// TIA Portal V16 export
// export: Created 2021-05-25T16:14:34.663981Z, ExportSetting WithDefaults, DisplayName Totally Integrated Automation Portal, DisplayVersion V16, DisplayName TIA Portal Version Control Interface, DisplayVersion V16, DisplayName TIA Portal Openness, DisplayVersion V16, DisplayName STEP 7 Professional, DisplayVersion V16, DisplayName STEP 7 Safety, DisplayVersion V16, DisplayName WinCC Unified SCADA Engineering System, DisplayVersion V16
DATA_BLOCK "ph_Helix_1_DB"   // DB310
VERSION : 0.1
// stored: AutoNumber false, DBAccessibleFromOPCUA true, InstanceOfName ph_Helix_1, InstanceOfType FB
"ph_Helix_1"
   // VAR_IN_OUT
   //    Y8_VijaLocev_Des : "udtDigitalValve";
   //    Y9_VijaStop_DesZad : "udtDigitalValve";
   //    Y2_VijaDesZad_Dvig : "udtDigitalValve";
   //    Y10_Centri_DesZad : "udtDigitalValve";
   //    Y3_VijaDesSpr_Dvig : "udtDigitalValve";
   //    Y11_Centri_DesSpr : "udtDigitalValve";
   //    Y12_VijaLocev_Lev : "udtDigitalValve";
   //    Y13_VijaStop_LevZad : "udtDigitalValve";
   //    Y4_VijaLevZad_Dvig : "udtDigitalValve";
   //    Y14_Centri_LevZad : "udtDigitalValve";
   //    Y5_VijaLevSpr_Dvig : "udtDigitalValve";
   //    Y15_Centri_LevSpr : "udtDigitalValve";
   //    Y16_VpenjanjeDna : "udtDigitalValve";
   //    M1_ZADAJ_LEVO : "udtMotor";
   //    M2_SPREDAJ_LEVO : "udtMotor";
   //    M1_ZADAJ_DESNO : "udtMotor";
   //    M2_SPREDAJ_DESNO : "udtMotor";
   //    VKLOP_M_TRAKA_VIJACNIKA : "udtMotor";
   // END_VAR
   // VAR RETAIN
   //    CurrentStep { ExternalAccessible := 'False'; ExternalVisible := 'False'; ExternalWritable := 'False'} : Int := 10;
   //    PhaseStatus { ExternalAccessible := 'False'; ExternalVisible := 'False'; ExternalWritable := 'False'} : Int := 5;
   // END_VAR
   // VAR
   //    AlarmPresent { ExternalAccessible := 'False'; ExternalVisible := 'False'; ExternalWritable := 'False'} : Bool := FALSE;
   //    InitPosition { ExternalAccessible := 'False'; ExternalVisible := 'False'; ExternalWritable := 'False'} : Bool := TRUE;
   //    StartCmd { ExternalAccessible := 'False'; ExternalVisible := 'False'; ExternalWritable := 'False'} : Bool := TRUE;
   //    AlarmPresentOLD { ExternalAccessible := 'False'; ExternalVisible := 'False'; ExternalWritable := 'False'} : Bool := FALSE;
   //    InitPositionOLD { ExternalAccessible := 'False'; ExternalVisible := 'False'; ExternalWritable := 'False'} : Bool := TRUE;
   //    IEC_TimerOnDly_1 { ExternalAccessible := 'False'; ExternalVisible := 'False'; ExternalWritable := 'False'} : TONR_TIME;
   //    IEC_TimerOnDly_2 { ExternalAccessible := 'False'; ExternalVisible := 'False'; ExternalWritable := 'False'} : TONR_TIME;
   //    IEC_TimerOnDly_3 { ExternalAccessible := 'False'; ExternalVisible := 'False'; ExternalWritable := 'False'} : TONR_TIME;
   //    IEC_TimerOnDly_4 { ExternalAccessible := 'False'; ExternalVisible := 'False'; ExternalWritable := 'False'} : TONR_TIME;
   //    IEC_TimerOnDly_5 { ExternalAccessible := 'False'; ExternalVisible := 'False'; ExternalWritable := 'False'} : TONR_TIME;
   //    IEC_TimerOnDly_6 { ExternalAccessible := 'False'; ExternalVisible := 'False'; ExternalWritable := 'False'} : TONR_TIME;
   //    IEC_TimerOnDly_7 { ExternalAccessible := 'False'; ExternalVisible := 'False'; ExternalWritable := 'False'} : TONR_TIME;
   //    IEC_TimerOnDly_8 { ExternalAccessible := 'False'; ExternalVisible := 'False'; ExternalWritable := 'False'} : TONR_TIME;
   //    IEC_TimerOnDly_9 { ExternalAccessible := 'False'; ExternalVisible := 'False'; ExternalWritable := 'False'} : TONR_TIME;
   //    IEC_TimerOnDly_10 { ExternalAccessible := 'False'; ExternalVisible := 'False'; ExternalWritable := 'False'} : TONR_TIME;
   //    IEC_TimerOnDly_ET_1 { ExternalAccessible := 'False'; ExternalVisible := 'False'; ExternalWritable := 'False'} : Time := T#0MS;
   //    IEC_TimerOnDly_ET_2 { ExternalAccessible := 'False'; ExternalVisible := 'False'; ExternalWritable := 'False'} : Time := T#0MS;
   //    IEC_TimerOnDly_ET_3 { ExternalAccessible := 'False'; ExternalVisible := 'False'; ExternalWritable := 'False'} : Time := T#0MS;
   //    IEC_TimerOnDly_ET_4 { ExternalAccessible := 'False'; ExternalVisible := 'False'; ExternalWritable := 'False'} : Time := T#0MS;
   //    IEC_TimerOnDly_ET_5 { ExternalAccessible := 'False'; ExternalVisible := 'False'; ExternalWritable := 'False'} : Time := T#0MS;
   //    IEC_TimerOnDly_ET_6 { ExternalAccessible := 'False'; ExternalVisible := 'False'; ExternalWritable := 'False'} : Time := T#0MS;
   //    IEC_TimerOnDly_ET_7 { ExternalAccessible := 'False'; ExternalVisible := 'False'; ExternalWritable := 'False'} : Time := T#0MS;
   //    IEC_TimerOnDly_ET_8 { ExternalAccessible := 'False'; ExternalVisible := 'False'; ExternalWritable := 'False'} : Time := T#0MS;
   //    IEC_TimerOnDly_ET_9 { ExternalAccessible := 'False'; ExternalVisible := 'False'; ExternalWritable := 'False'} : Time := T#0MS;
   //    IEC_TimerOnDly_ET_10 { ExternalAccessible := 'False'; ExternalVisible := 'False'; ExternalWritable := 'False'} : Time := T#0MS;
   //    IEC_TimerOnDly_DN_1 { ExternalAccessible := 'False'; ExternalVisible := 'False'; ExternalWritable := 'False'} : Bool := FALSE;
   //    IEC_TimerOnDly_DN_2 { ExternalAccessible := 'False'; ExternalVisible := 'False'; ExternalWritable := 'False'} : Bool := FALSE;
   //    IEC_TimerOnDly_DN_3 { ExternalAccessible := 'False'; ExternalVisible := 'False'; ExternalWritable := 'False'} : Bool := FALSE;
   //    IEC_TimerOnDly_DN_4 { ExternalAccessible := 'False'; ExternalVisible := 'False'; ExternalWritable := 'False'} : Bool := FALSE;
   //    IEC_TimerOnDly_DN_5 { ExternalAccessible := 'False'; ExternalVisible := 'False'; ExternalWritable := 'False'} : Bool := FALSE;
   //    IEC_TimerOnDly_DN_6 { ExternalAccessible := 'False'; ExternalVisible := 'False'; ExternalWritable := 'False'} : Bool := FALSE;
   //    IEC_TimerOnDly_DN_7 { ExternalAccessible := 'False'; ExternalVisible := 'False'; ExternalWritable := 'False'} : Bool := FALSE;
   //    IEC_TimerOnDly_DN_8 { ExternalAccessible := 'False'; ExternalVisible := 'False'; ExternalWritable := 'False'} : Bool := FALSE;
   //    IEC_TimerOnDly_DN_9 { ExternalAccessible := 'False'; ExternalVisible := 'False'; ExternalWritable := 'False'} : Bool := FALSE;
   //    IEC_TimerOnDly_DN_10 { ExternalAccessible := 'False'; ExternalVisible := 'False'; ExternalWritable := 'False'} : Bool := FALSE;
   //    LeftLegIndex { ExternalAccessible := 'False'; ExternalVisible := 'False'; ExternalWritable := 'False'} : Int := 2;
   //    RightLegIndex { ExternalAccessible := 'False'; ExternalVisible := 'False'; ExternalWritable := 'False'} : Int := 2;
   //    LeftLegsArrayIndex { ExternalAccessible := 'False'; ExternalVisible := 'False'; ExternalWritable := 'False'} : Array[1..6] of Bool;
   //    RightLegsArrayIndex { ExternalAccessible := 'False'; ExternalVisible := 'False'; ExternalWritable := 'False'} : Array[1..6] of Bool;
   //    ButtomFasting_Activated { ExternalAccessible := 'False'; ExternalVisible := 'False'; ExternalWritable := 'False'} : Bool := TRUE;
   //    Helix_Activated { ExternalAccessible := 'False'; ExternalVisible := 'False'; ExternalWritable := 'False'} : Bool := FALSE;
   // END_VAR
   // VAR RETAIN
   //    DlyToFinishButtonFasten { S7_SetPoint := 'True'} : Int := 2;
   // END_VAR
   // VAR
   //    MovingUPDOWN_Activated { ExternalAccessible := 'False'; ExternalVisible := 'False'; ExternalWritable := 'False'} : Bool := FALSE;
   //    MoveUPDOWN_LevoSpredaj { ExternalAccessible := 'False'; ExternalVisible := 'False'; ExternalWritable := 'False'} : Bool := FALSE;
   //    MoveUPDOWN_LevoZadaj { ExternalAccessible := 'False'; ExternalVisible := 'False'; ExternalWritable := 'False'} : Bool := FALSE;
   //    MoveUPDOWN_DESNOSpredaj { ExternalAccessible := 'False'; ExternalVisible := 'False'; ExternalWritable := 'False'} : Bool := FALSE;
   //    MoveUPDOWN_DESNOZadaj { ExternalAccessible := 'False'; ExternalVisible := 'False'; ExternalWritable := 'False'} : Bool := FALSE;
   // END_VAR
   // VAR RETAIN
   //    DlyToRotateOpposite { S7_SetPoint := 'True'} : Int := 10;
   //    WaitTimeBeforeMoveDown { S7_SetPoint := 'True'} : Int := 2;
   // END_VAR
   // VAR
   //    WaitLevoSpredaj { ExternalAccessible := 'False'; ExternalVisible := 'False'; ExternalWritable := 'False'} : Bool := FALSE;
   //    WaitLevoZadaj { ExternalAccessible := 'False'; ExternalVisible := 'False'; ExternalWritable := 'False'} : Bool := FALSE;
   //    WaitDesnoSpredaj { ExternalAccessible := 'False'; ExternalVisible := 'False'; ExternalWritable := 'False'} : Bool := FALSE;
   //    WaitDesnoZadaj { ExternalAccessible := 'False'; ExternalVisible := 'False'; ExternalWritable := 'False'} : Bool := FALSE;
   //    FOTOCELICA_LOC_TRAK_LEVO1_Latch { ExternalAccessible := 'False'; ExternalVisible := 'False'; ExternalWritable := 'False'} : Bool := FALSE;
   //    FOTOCELICA_LOC_TRAK_LEVO2_Latch { ExternalAccessible := 'False'; ExternalVisible := 'False'; ExternalWritable := 'False'} : Bool := FALSE;
   //    FOTOCELICA_LOC_TRAK_DESNO1_Latch { ExternalAccessible := 'False'; ExternalVisible := 'False'; ExternalWritable := 'False'} : Bool := FALSE;
   //    FOTOCELICA_LOC_TRAK_DESNO2_Latch { ExternalAccessible := 'False'; ExternalVisible := 'False'; ExternalWritable := 'False'} : Bool := FALSE;
   // END_VAR
   // VAR RETAIN
   //    WEndTimeToRemovePlate { S7_SetPoint := 'True'} : Int := 2;
   // END_VAR
   // VAR
   //    LeftLegIndexOLD { ExternalAccessible := 'False'; ExternalVisible := 'False'; ExternalWritable := 'False'} : Int := 2;
   //    RightLegIndexOLD { ExternalAccessible := 'False'; ExternalVisible := 'False'; ExternalWritable := 'False'} : Int := 2;
   //    StartReleaseTimer1 { ExternalAccessible := 'False'; ExternalVisible := 'False'; ExternalWritable := 'False'} : Bool := FALSE;
   //    StartReleaseTimer2 { ExternalAccessible := 'False'; ExternalVisible := 'False'; ExternalWritable := 'False'} : Bool := FALSE;
   //    FOTOCELICA_LEVO_SPREDAJ_LATCH { ExternalAccessible := 'False'; ExternalVisible := 'False'; ExternalWritable := 'False'} : Bool := TRUE;
   //    FOTOCELICA_LEVO_ZADAJ_LATCH { ExternalAccessible := 'False'; ExternalVisible := 'False'; ExternalWritable := 'False'} : Bool := TRUE;
   //    FOTOCELICA_DESNO_SPREDAJ_LATCH { ExternalAccessible := 'False'; ExternalVisible := 'False'; ExternalWritable := 'False'} : Bool := TRUE;
   //    FOTOCELICA_DESNO_ZADAJ_LATCH { ExternalAccessible := 'False'; ExternalVisible := 'False'; ExternalWritable := 'False'} : Bool := TRUE;
   // END_VAR
   // VAR RETAIN
   //    DlyToStartButtomFasten { S7_SetPoint := 'True'} : Int := 10;
   // END_VAR
   // VAR
   //    EndLevoSpredaj { ExternalAccessible := 'False'; ExternalVisible := 'False'; ExternalWritable := 'False'} : Bool := FALSE;
   //    EndLevoZadaj { ExternalAccessible := 'False'; ExternalVisible := 'False'; ExternalWritable := 'False'} : Bool := FALSE;
   //    EndDesnoSpredaj { ExternalAccessible := 'False'; ExternalVisible := 'False'; ExternalWritable := 'False'} : Bool := FALSE;
   //    EndDesnoZadaj { ExternalAccessible := 'False'; ExternalVisible := 'False'; ExternalWritable := 'False'} : Bool := FALSE;
   // END_VAR
   // VAR RETAIN
   //    DlyToInitRunTrakVijac { ExternalAccessible := 'False'; ExternalVisible := 'False'; ExternalWritable := 'False'; S7_SetPoint := 'True'} : Int := 20;
   // END_VAR
   // VAR
   //    LegsReadyOnPosToHelix { ExternalAccessible := 'False'; ExternalVisible := 'False'; ExternalWritable := 'False'} : Bool := FALSE;
   //    VpenjanjeDnaActived { ExternalAccessible := 'False'; ExternalVisible := 'False'; ExternalWritable := 'False'} : Bool := FALSE;
   // END_VAR
   // VAR RETAIN
   //    RegimeHelix { S7_SetPoint := 'True'} : Bool := TRUE;
   //    TotalButtomPlateCounter : UDInt := 4;
   // END_VAR
   // VAR
   //    DetectStartButtom { ExternalAccessible := 'False'; ExternalVisible := 'False'; ExternalWritable := 'False'} : Bool := FALSE;
   //    InsertNewButtom { ExternalAccessible := 'False'; ExternalVisible := 'False'; ExternalWritable := 'False'} : USInt := 1;
   // END_VAR
   // VAR RETAIN
   //    TimeoutToEndHelix { ExternalAccessible := 'False'; ExternalVisible := 'False'; ExternalWritable := 'False'; S7_SetPoint := 'True'} : UInt := 80;
   // END_VAR
   // VAR
   //    FirstButtom { ExternalAccessible := 'False'; ExternalVisible := 'False'; ExternalWritable := 'False'} : Bool := FALSE;
   // END_VAR
BEGIN
   IEC_TimerOnDly_1.PT := T#0MS;
   IEC_TimerOnDly_1.IN := FALSE;
   IEC_TimerOnDly_2.PT := T#0MS;
   IEC_TimerOnDly_2.IN := FALSE;
   IEC_TimerOnDly_3.PT := T#0MS;
   IEC_TimerOnDly_3.IN := FALSE;
   IEC_TimerOnDly_4.PT := T#0MS;
   IEC_TimerOnDly_4.IN := FALSE;
   IEC_TimerOnDly_5.PT := T#0MS;
   IEC_TimerOnDly_5.IN := FALSE;
   IEC_TimerOnDly_6.PT := T#0MS;
   IEC_TimerOnDly_6.IN := FALSE;
   IEC_TimerOnDly_7.PT := T#0MS;
   IEC_TimerOnDly_7.IN := FALSE;
   IEC_TimerOnDly_8.PT := T#0MS;
   IEC_TimerOnDly_8.IN := FALSE;
   IEC_TimerOnDly_9.PT := T#0MS;
   IEC_TimerOnDly_9.IN := FALSE;
   IEC_TimerOnDly_10.PT := T#0MS;
   IEC_TimerOnDly_10.IN := FALSE;
   LeftLegsArrayIndex[1..2] := TRUE;
   LeftLegsArrayIndex[3..6] := FALSE;
   RightLegsArrayIndex[1..2] := TRUE;
   RightLegsArrayIndex[3..6] := FALSE;
END_DATA_BLOCK
